//////////////////////////////////////////////////////////////////
// Structure For PDL. Main Operating Data to be saved (ex: OPC) //  
//////////////////////////////////////////////////////////////////

TYPE SUBHV :
STRUCT
	// Substation Data
	
	MesAlarmCode				: WORD ; (* (NA) Internal Akuo AlarmCode 	*) 
 	MesWarningCode				: WORD ; (* (NA) Internal Akuo WarningCode  *)
	MesEventCode				: WORD ; (* (NA) Internal Akuo EventCode 	*)
	
END_STRUCT
END_TYPE

(* stored: Version 1.1.0.1, ProductVersion 3.1.4024.6
   DUT SUBHV: Id {5714af5e-b1a5-428f-8412-8e82bd391c10} *)
